# EPICS substitutions: ek9000App/Db/EL4122.substitutions
file EL4122.template
{       pattern
        {
                TERMINAL,

        }
        {
        }
}
